TYPE T_DEVICE_ID : STRING; END_TYPE

(* stored: Version 1.1.0.1, ProductVersion 3.1.4026.18
   DUT T_DEVICE_ID: Id {833d1cb0-98f7-0c08-14a5-7ad95f336149} *)
